{attribute 'GeneratedUsingTerminal: EJ2521-0224-0016'}
{attribute addProperty BoxType "EJ2521-0224-0016"}
{attribute addProperty Id "Target_counter_valueAT %Q*UINT2"}
{attribute addProperty CRC "1547018109"}
{attribute addProperty Size "2"}
TYPE PTO_Target_compact_5C359F7D :
STRUCT
	{attribute addProperty Name "Target_counter_value"}
	Target_counter_value AT %Q* : UINT;
END_STRUCT
END_TYPE

(* stored: Version 1.2.0.0, ProductVersion 3.1.4024.9
   DUT PTO_Target_compact_5C359F7D: Id {eda2e275-a137-4085-b81e-1e01ed2851a1} *)
